TYPE ST_EjectorParameters :
STRUCT
	ejectPositionPass 	: LREAL; // := 100;
	ejectPositionHome 	: LREAL; // := 50;
	ejectPositionFail 	: LREAL; // := 0;
	ejectVelocity		: LREAL; // := 20;
END_STRUCT
END_TYPE

(* stored: Version 1.1.0.1, ProductVersion 3.1.4024.9
   DUT ST_EjectorParameters: Id {4d391966-b6d6-4584-b4cc-e939f59249b6} *)
